Universal Robots PolyScope program: robolab_c3_13.urp

Program robolab_c3_13 (installation=default directory=/programs createdIn=3.14.3.1031232 lastSavedIn=3.15.8.106339 robotSerialNumber=2020330428)
Calibrated DH parameters: a=[0.000029, -0.241913, -0.128453, -0.000049, -0.000012, 0]; d=[0.151842, -4.082088, 33.504745, -29.309875, 0.08529, 0.082285]; alpha=[1.571059, -0.006644, 0.005794, 1.571984, -1.571997, 0]; deltaTheta=[-0.000032, 0.111537, 0.813391, -0.924919, 0.000036, 0.000016]
Robot Program (runOnlyOnce=false)
  URCap External Control (External Control, FZI Research Center for Information Technology)
